// TIA Portal V20 export
TYPE "LConSMC_typePIDControllerIn"
// stored: Access Published
   STRUCT
      enable : Bool := FALSE;   // TRUE: Funktionsbaustein aktivieren / TRUE: Enable function block
      reset : Bool := FALSE;   // TRUE: Funktionsbaustein zurücksetzen / TRUE: Reset function block
      setpointValue : LReal := 0.0;   // [-] Sollwert / [-] Setpoint
      actualValue : LReal := 0.0;   // [-] Istwert / [-] Actual value
      preControl : LReal := 0.0;   // Reglervorsteuerung / Controler pre control value
      propGain : LReal := 2.0;   // Proportionalverstärkung Ein Wert von 0 deaktiviert den P-Anteil / Proportional gain. A value of 0 disables the P-part
      integTime : LReal := 999.0;   // [ms] Integrationszeitkonstante Ein Wert von 0 deaktiviert den I-Anteil / [ms] Time constant for integrator. A value of 0 disables the I-part
      derivTime : LReal := 0.0;   // [ms] Differentationszeitkonstante Ein Wert von 0 deaktiviert den D-Anteil / [ms] Time constant for differentiator. A value of 0 disables the D-part
      filterTime : LReal := 10.0;   // [ms] PT1 - Istwertfilter Ein Wert von 0 deaktiviert den Filter / [ms] PT1- Filter for actual value. A value of 0 disables the filter
      upperLimit : LReal := 100.0;   // Oberer Grenze des Reglerausgangs / Upper limit of the controller output
      lowerLimit : LReal := 0.0;   // Untere Grenze des Reglerausgangs / Lower limit of the controller output
      intSetValue : LReal := 0.0;   // Setzwert des Integrators (wenn "setIntChannel" = TRUE) / Integrator set value (if "setIntChannel" = TRUE)
      holdIntChannel : Bool := FALSE;   // TRUE: Integrator wird angehalten / TRUE: Integrator is hold
      setIntChannel : Bool := FALSE;   // TRUE: Der Wert des Integrators wird auf "intSetValue" gesetzt / TRUE: The output of the integrator is set to "intSetValue"
      controlMode : Bool := FALSE;   // TRUE: D-Komponente aktiv im Istwert-Pfad FALSE: D-Komponente aktiv in der Reglerabweichung / TRUE: D component active in actual value branch FALSE: D component in controller deviation
      deadBand { ExternalAccessible := 'False'; ExternalVisible := 'False'; ExternalWritable := 'False'} : LReal := 0.0;   // Breite des Totbandes (symmetrisch). Ein Wert von 0 deaktiviert das Totband / Value of the dead band (symmetrical). A value of 0 disables the deadband
      actualValueFactor : LReal := 1.0;   // Multiplikativer Skalierungsfaktor des Istwertes / Multiplicative scaling of the actual value
      actualValueOffset : LReal := 0.0;   // Additiver Skalierungsfaktor des Istwertes / Additive scaling of the actual value
      outValueFactor : LReal := 1.0;   // Multiplikativer Skalierungsfaktor des Reglerausgangs / Multiplicative scaling of the controller output
      outValueOffset : LReal := 0.0;   // Additiver Skalierungsfaktor des Reglerausgangs / Additive scaling of the controller output
      tCycle : Real := 0.0;   // [ms] Zykluszeit in der der Baustein aufgerufen wird / [ms] Cycle time the function block is called
   END_STRUCT;
END_TYPE
